// TIA Portal V18 export
TYPE "UDT_V90_Axis_Positions"
   STRUCT
      Position { S7_SetPoint := 'True'} : Array[1..20] of "UDT_Motion_Point_V90";
   END_STRUCT;
END_TYPE
